(* PLC project Tc2_Utilities.SYSTEMTIME_TO_ISO8601 Demo, tc3-libraries-kb TwinCAT 3.1 *)
(* stored: creationDateTime 2026-05-10T12:00:00, modificationDateTime 2026-05-10T12:00:00 *)

PROGRAM P_Demo_SYSTEMTIME_TO_ISO8601
  VAR
    rResult : STRING;  (* SYSTEMTIME_TO_ISO8601 的返回值 *)
    bRun : BOOL;  (* 触发一次调用 *)
    stIn : TIMESTRUCT;  (* 测试用本地变量 *)
  END_VAR

            // ============================================================
// Tc2_Utilities.SYSTEMTIME_TO_ISO8601 演示程序（FUNCTION）
// ============================================================
// 验证步骤：
//   1. 引用 Tc2_Utilities（及类型所在依赖库 Tc2_System / Tc2_Standard）
//   2. 编译 + 登录
//   3. 强制 bRun := TRUE 一个周期
//   4. 观察 rResult 应为 '2024-01-01T13:00:00.000+01:00'
// ============================================================

stIn.wYear := 2024; stIn.wMonth := 1; stIn.wDay := 1; stIn.wHour := 12;
IF bRun THEN
    rResult := SYSTEMTIME_TO_ISO8601(stIn, 60, FALSE, 3);
    bRun := FALSE;
END_IF;

          
END_PROGRAM
